TYPE
    ST_HMI_ShippingArea :
    STRUCT
        //提供新的馬達
    END_STRUCT
END_TYPE

(* stored: Version 1.1.0.1, ProductVersion 3.1.4024.13
   DUT ST_HMI_ShippingArea: Id {fc509919-1459-4ef2-8600-ff37a539f56a} *)
